(* IEC 61131-3 sources: CODESYS-IO-Visualization/CODESYS-IO-Visualization.fbsproj/Subs/IO/Opto22, 5 files *)

(* ---- IO_StatusCodeToString.prg.st ---- *)
PROGRAM IO_StatusCodeToString

VAR_IN_OUT
	Data: Channel_UDT;
END_VAR

Data.StatusCode := WORD_TO_DINT(Data.ValueStatus);

IF (Data.ValueStatus = 0) THEN
	Data.StatusString := "";
	RETURN;
END_IF;

IF (Data.ValueStatus.0) THEN
	Data.StatusString := "Out of Range";
ELSE
	Data.StatusString := "Failed";
END_IF;

(* ---- Module_Opto.prg.st ---- *)
PROGRAM Module_Opto

VAR_IN_OUT
	Rack: Rack_Opto_RIO_UDT;
	Module: Module_Opto_UDT;
END_VAR

VAR
	TempStat: DWORD;
	i: INT;
END_VAR

IF (Module.CI OR (NOT Module.InUse) OR Rack.CI OR (NOT Rack.InUse)) THEN
	Module.Status := -1;
	Module.StatusString := "Control Inhibit or Disabled";
ELSE
	IF (Module.Module_IO <> 0) THEN
		Module.IsRIO := FALSE;

		IF (Module.SimulationEnable AND Simulation.SimulationEnable) THEN
			Module.Status := Module.Simulator.odiStatusCode;
			Module.StatusString := Module.Simulator.osStatusCode;
		ELSE
			Module.ModuleTypeId := Module.Module_IO^._pModType;
			Module.ModuleConfigFailed := Module.Module_IO^._bConfigureModuleFailed;
			Module.ModuleConfigFound := Module.Module_IO^._bConfigureModuleFound;
			Module.ModuleMissing := Module.Module_IO^._bMissingModule;
			Module.Deactivated := Module.Module_IO^._bDeactivated;
			Module.NumberOfChannels := Module.Module_IO^._udiNumChannels;
		END_IF;
	ELSIF (Module.RIO_IO <> 0) THEN
		Module.IsRIO := TRUE;

		IF (Module.SimulationEnable AND Simulation.SimulationEnable) THEN
			Module.Status := Module.Simulator.odiStatusCode;
			Module.StatusString := Module.Simulator.osStatusCode;
		ELSE
			Module.ModuleTypeId := 0;
			Module.ModuleConfigFailed := NOT Module.RIO_IO^.xConfigFinished;
			Module.ModuleConfigFound := Module.RIO_IO^.xConfigFinished;
			Module.ModuleMissing := Module.RIO_IO^.xError;
			Module.Deactivated := FALSE;
			Module.NumberOfChannels := 10;
		END_IF;
	ELSE
		Module.Status := 255;
		Module.StatusString := "Invalid Pointer for IO Module";
	END_IF;

	IF (Module.Module_IO = 0 AND Module.RIO_IO = 0) THEN
		Module.Status := 255;
		Module.StatusString := "Invalid Pointer for IO Module";
	ELSE
		TempStat := 0;
		TempStat.0 := Module.Deactivated;
		TempStat.1 := Module.ModuleConfigFailed;
		TempStat.2 := Module.ModuleMissing;
		TempStat.3 := Module.ModuleMissing;

		Module.Status := DWORD_TO_DINT(TempStat);

		CASE TempStat OF
			0:
				Module.StatusString := "";
			1:
				Module.StatusString := "Module Deactivated";
			2..3:
				Module.StatusString := "Module Configuration Failure";
			4..7:
				Module.StatusString := "Module Not Found";
			8..15:
				Module.StatusString := "Module Missing";
		ELSE
				Module.StatusString := "Module Failed";
		END_CASE;
	END_IF;
END_IF;

Module.Failed.Enable := Module.InUse AND Rack.InUse AND (NOT Module.CI) AND (NOT Rack.CI);
Module.Failed.Value := (Module.Status > 0);
AlarmDigital(alarm := Module.Failed);

(* ---- ProcessModuleIO_Opto.prg.st ---- *)
PROGRAM ProcessModuleIO_Opto

VAR_IN_OUT
	Rack: Rack_Opto_RIO_UDT;
	Module: Module_Opto_UDT;
END_VAR

VAR
	i: INT;
END_VAR

FOR i := 0 TO Lib_GVL.MaxPointCount DO
	CASE Module.Channels[i].ChannelType OF
		IOChannelType.ctAO:
			IOA_Output(Data := Module.Channels[i], ModuleStatus := Module.Status, ModuleCI := Module.CI);

		IOChannelType.ctDO:
			IOD_Output(Data := Module.Channels[i], ModuleStatus := Module.Status, ModuleCI := Module.CI);
	END_CASE;

	CASE Module.Channels[i].ChannelType OF
		IOChannelType.ctAI:
			Module.Channels[i].ValueRawAnalog := Module.IO[i].Ana;
			Module.Channels[i].ValueStatus.0 := FPU.IsRealNaN(Module.IO[i].Ana) OR
				(Module.Channels[i].ValueRawAnalog > Module.Channels[i].ZeroRaw + (Module.Channels[i].SpanRaw * 1.04)) OR
				(Module.Channels[i].ValueRawAnalog < Module.Channels[i].ZeroRaw - (Module.Channels[i].SpanRaw * 0.04));

		IOChannelType.ctAO:
			Module.IO[i].Ana := Module.Channels[i].ValueRawAnalogOut;
			Module.Channels[i].ValueRawAnalog := Module.IO[i].Ana;
			Module.Channels[i].ValueStatus.0 :=
				(Module.Channels[i].ValueRawAnalog > Module.Channels[i].ZeroRaw + (Module.Channels[i].SpanRaw * 1.04)) OR
				(Module.Channels[i].ValueRawAnalog < Module.Channels[i].ZeroRaw - (Module.Channels[i].SpanRaw * 0.04));

		IOChannelType.ctDI:
			Module.Channels[i].ValueRawDigital := Module.IO[i].Dig;
			Module.Channels[i].ValueStatus := 0;

		IOChanneltype.ctDO:
			Module.IO[i].Dig := Module.Channels[i].ValueRawDigitalOut;
			Module.Channels[i].ValueRawDigital := Module.IO[i].Dig;
			Module.Channels[i].ValueStatus := 0;
	END_CASE;

	CASE Module.Channels[i].ChannelType OF
		IOChannelType.ctAI:
			IOA_Input(Data := Module.Channels[i], ModuleStatus := Module.Status, ModuleCI := Module.CI);

		IOChanneltype.ctDI:
			IOD_Input(Data := Module.Channels[i], ModuleStatus := Module.Status, ModuleCI := Module.CI);
	END_CASE;
END_FOR;

(* ---- ProcessRackIO_Opto.prg.st ---- *)
PROGRAM ProcessRackIO_Opto

VAR_IN_OUT
	Rack: Rack_Opto_RIO_UDT;
END_VAR

VAR
	i: INT;
END_VAR

FOR i := 0 TO Lib_GVL.MaxModuleCount DO
	ProcessModuleIO_Opto(Rack := Rack, Module := Rack.Modules[i]);
END_FOR;

(* ---- Rack_Opto_RIO.prg.st ---- *)
{attribute "analysis" := "-90"}PROGRAM Rack_Opto_RIO

VAR_IN_OUT
	Rack: Rack_Opto_RIO_UDT;
END_VAR

VAR
	TempStat: DWORD;
	i: INT;
END_VAR

IF (Rack.CI OR (NOT Rack.InUse)) THEN
	Rack.Status := -1;
	Rack.StatusString := "Control Inhibit or Disabled";
	ProcessModules();
	RETURN;
END_IF;

IF (Rack.Rack_IO = 0) THEN
	Rack.Status := 255;
	Rack.StatusString := "Invalid Pointer for IO Rack";
	ProcessModules();
	RETURN;
END_IF;

Rack.Deactivated := FALSE;
Rack.ConfigFinished := TRUE;
Rack.ConfigStepError := FALSE;
Rack.Error := FALSE;
Rack.IpAddr := "Unknown";
Rack.DiagString := "";

TempStat := 0;
TempStat.0 := Rack.Deactivated;
TempStat.1 := Rack.Error;
TempStat.2 := Rack.ConfigStepError;
TempStat.3 := NOT Rack.ConfigFinished;

Rack.Status := DWORD_TO_DINT(TempStat);
Rack.StatusString := Rack.DiagString;

ProcessModules();
